TYPE AX5000_P_0453 :
STRUCT
	Current_controller_status_word:UINT;
END_STRUCT
END_TYPE

(* stored: Version 1.1.0.1, ProductVersion 3.1.4024.3
   DUT AX5000_P_0453: Id {8949e3c2-c04f-45dd-833d-1ee5c52729d7} *)
